(* Logix 5000 project; controller SX_V040001_C001 vendor 1 type 14 code 77 rev 16.22; software revision 16.04; part 6 of 35 *)
(* tags used below, declared in another part *)
   ALARM_BITS : INT[10];
   ALL_KINDS : INT[90];
   Basic : INT;
   G_DInput : DINT[3];
   G_DOutput : DINT[3];
   m_alarm_exist : BOOL;
   m_notstop : BOOL;
   METERING : INT[44];
   PARAMETER : INT[501];
   T_MET10_END : TIMER;
   T_MET11_END : TIMER;
   T_MET6_END : TIMER;
   T_MET7_END : TIMER;
   T_MET8_END : TIMER;
   T_MET9_END : TIMER;
   T_MET_VALVE_10 : TIMER;
   T_MET_VALVE_11 : TIMER;
   T_MET_VALVE_12 : TIMER;
   T_MET_VALVE_6 : TIMER;
   T_MET_VALVE_7 : TIMER;
   T_MET_VALVE_8 : TIMER;
   T_MET_VALVE_9 : TIMER;
   Z41 : COUNTER;
   Z42 : COUNTER;
   Z43 : COUNTER;
   Z44 : COUNTER;
   Z45 : COUNTER;
   Z46 : COUNTER;
   Z47 : COUNTER;
   Z48 : COUNTER;
   Z49 : COUNTER;
   Z50 : COUNTER;
(* MainProgram, continued *)

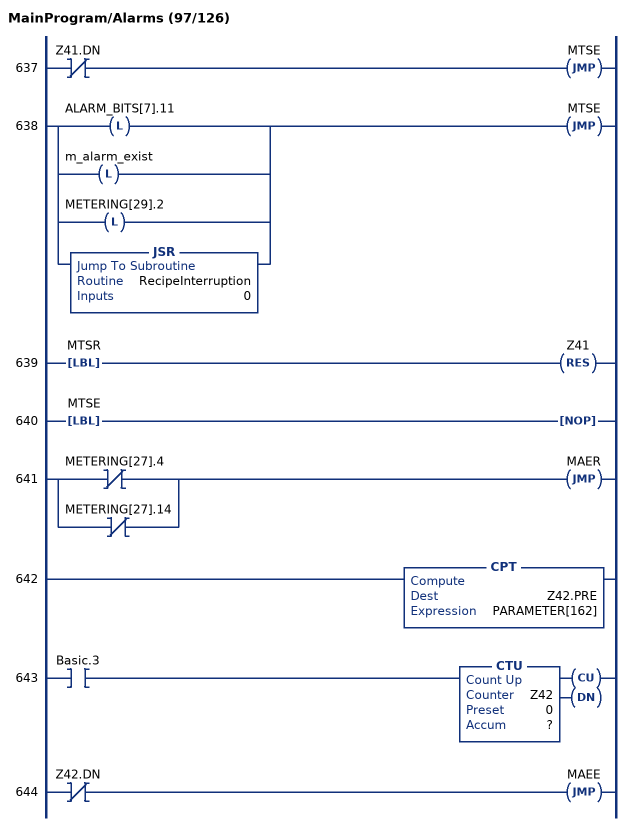
   [picture p118: MainProgram/Alarms rungs 637-644]
   637: XIO(Z41.DN)JMP(MTSE);
   638: [OTL(ALARM_BITS[7].11) ,OTL(m_alarm_exist) ,OTL(METERING[29].2) ,JSR(RecipeInterruption,0) ]JMP(MTSE);
   639: LBL(MTSR)RES(Z41);
   640: LBL(MTSE)NOP();
   641: [XIO(METERING[27].4) ,XIO(METERING[27].14) ]JMP(MAER);
   642: CPT(Z42.PRE,PARAMETER[162]);
   643: XIC(Basic.3)CTU(Z42,?,?);
   644: XIO(Z42.DN)JMP(MAEE);
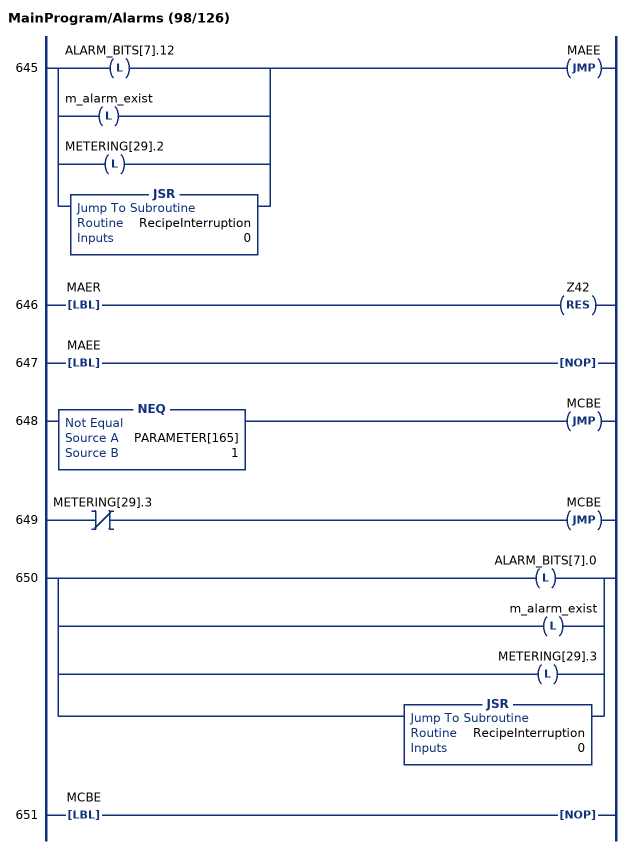
   645: [OTL(ALARM_BITS[7].12) ,OTL(m_alarm_exist) ,OTL(METERING[29].2) ,JSR(RecipeInterruption,0) ]JMP(MAEE);
   646: LBL(MAER)RES(Z42);
   647: LBL(MAEE)NOP();
   648: NEQ(PARAMETER[165],1)JMP(MCBE);
   649: XIO(METERING[29].3)JMP(MCBE);
   650: [OTL(ALARM_BITS[7].0) ,OTL(m_alarm_exist) ,OTL(METERING[29].3) ,JSR(RecipeInterruption,0) ];
   651: LBL(MCBE)NOP();
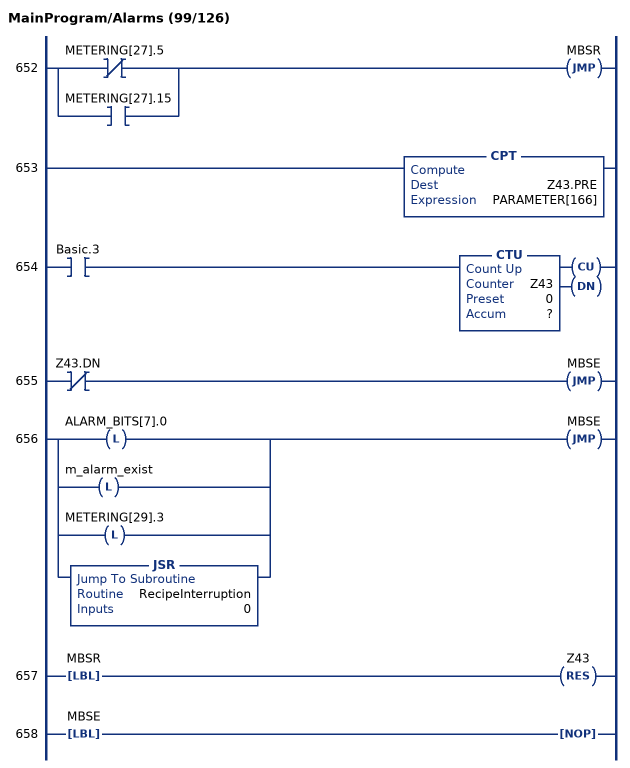
   652: [XIO(METERING[27].5) ,XIC(METERING[27].15) ]JMP(MBSR);
   653: CPT(Z43.PRE,PARAMETER[166]);
   654: XIC(Basic.3)CTU(Z43,?,?);
   655: XIO(Z43.DN)JMP(MBSE);
   656: [OTL(ALARM_BITS[7].0) ,OTL(m_alarm_exist) ,OTL(METERING[29].3) ,JSR(RecipeInterruption,0) ]JMP(MBSE);
   657: LBL(MBSR)RES(Z43);
   658: LBL(MBSE)NOP();
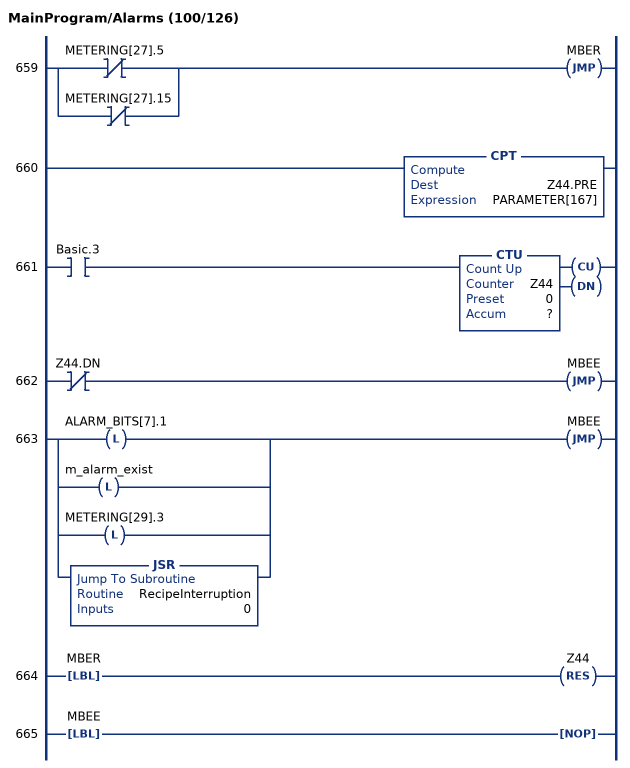
   659: [XIO(METERING[27].5) ,XIO(METERING[27].15) ]JMP(MBER);
   660: CPT(Z44.PRE,PARAMETER[167]);
   661: XIC(Basic.3)CTU(Z44,?,?);
   662: XIO(Z44.DN)JMP(MBEE);
   663: [OTL(ALARM_BITS[7].1) ,OTL(m_alarm_exist) ,OTL(METERING[29].3) ,JSR(RecipeInterruption,0) ]JMP(MBEE);
   664: LBL(MBER)RES(Z44);
   665: LBL(MBEE)NOP();
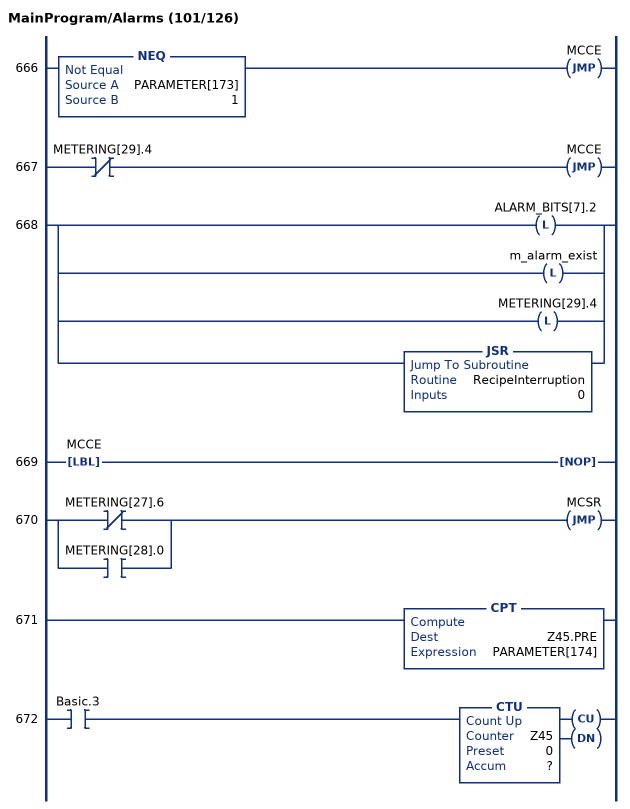
   666: NEQ(PARAMETER[173],1)JMP(MCCE);
   667: XIO(METERING[29].4)JMP(MCCE);
   668: [OTL(ALARM_BITS[7].2) ,OTL(m_alarm_exist) ,OTL(METERING[29].4) ,JSR(RecipeInterruption,0) ];
   669: LBL(MCCE)NOP();
   670: [XIO(METERING[27].6) ,XIC(METERING[28].0) ]JMP(MCSR);
   671: CPT(Z45.PRE,PARAMETER[174]);
   672: XIC(Basic.3)CTU(Z45,?,?);
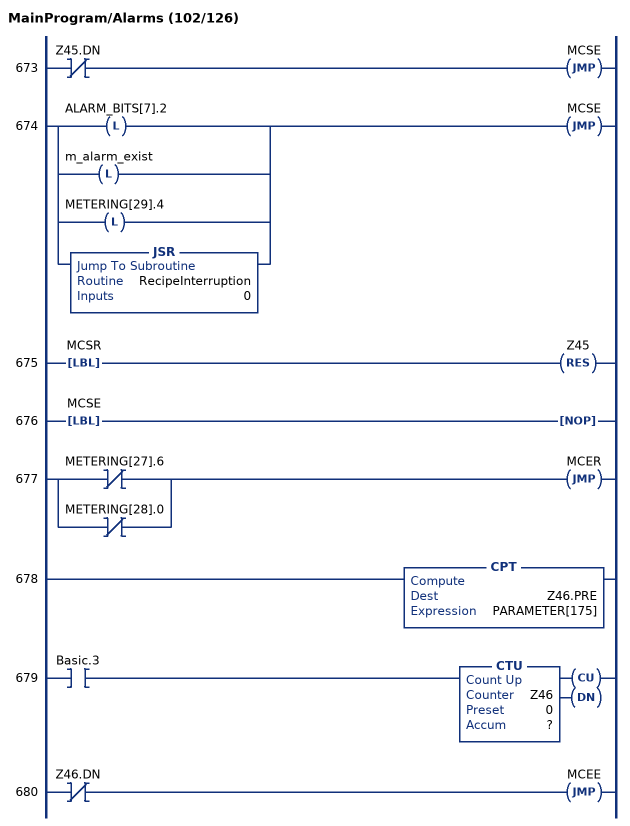
   673: XIO(Z45.DN)JMP(MCSE);
   674: [OTL(ALARM_BITS[7].2) ,OTL(m_alarm_exist) ,OTL(METERING[29].4) ,JSR(RecipeInterruption,0) ]JMP(MCSE);
   675: LBL(MCSR)RES(Z45);
   676: LBL(MCSE)NOP();
   677: [XIO(METERING[27].6) ,XIO(METERING[28].0) ]JMP(MCER);
   678: CPT(Z46.PRE,PARAMETER[175]);
   679: XIC(Basic.3)CTU(Z46,?,?);
   680: XIO(Z46.DN)JMP(MCEE);
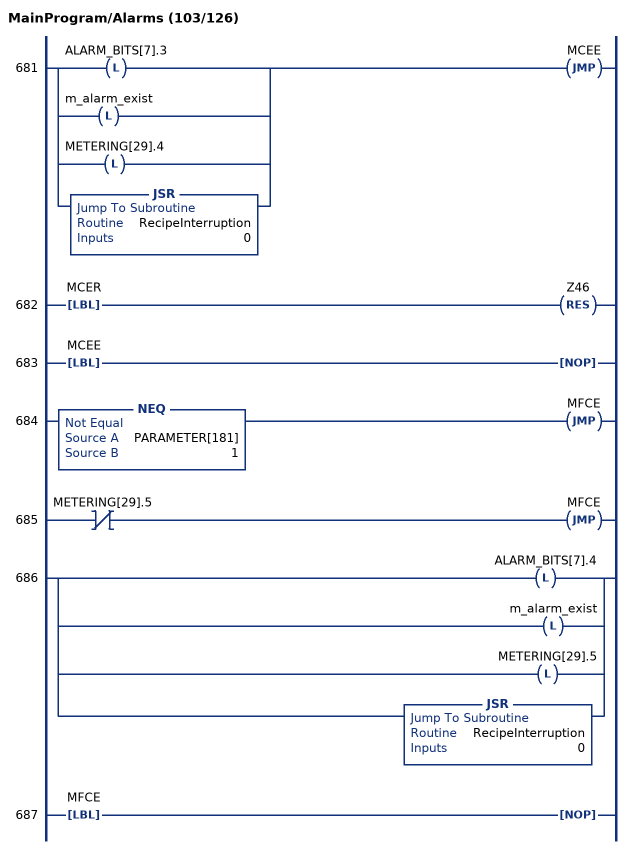
   681: [OTL(ALARM_BITS[7].3) ,OTL(m_alarm_exist) ,OTL(METERING[29].4) ,JSR(RecipeInterruption,0) ]JMP(MCEE);
   682: LBL(MCER)RES(Z46);
   683: LBL(MCEE)NOP();
   684: NEQ(PARAMETER[181],1)JMP(MFCE);
   685: XIO(METERING[29].5)JMP(MFCE);
   686: [OTL(ALARM_BITS[7].4) ,OTL(m_alarm_exist) ,OTL(METERING[29].5) ,JSR(RecipeInterruption,0) ];
   687: LBL(MFCE)NOP();
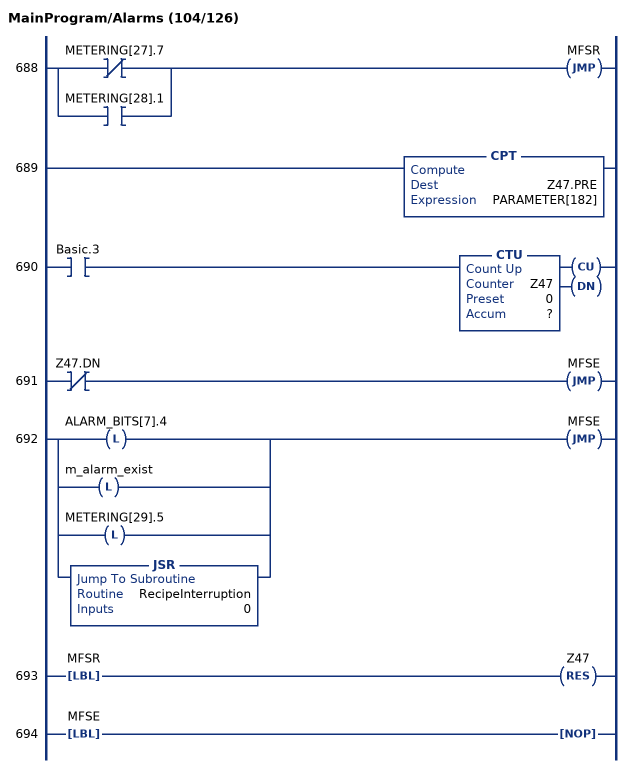
   688: [XIO(METERING[27].7) ,XIC(METERING[28].1) ]JMP(MFSR);
   689: CPT(Z47.PRE,PARAMETER[182]);
   690: XIC(Basic.3)CTU(Z47,?,?);
   691: XIO(Z47.DN)JMP(MFSE);
   692: [OTL(ALARM_BITS[7].4) ,OTL(m_alarm_exist) ,OTL(METERING[29].5) ,JSR(RecipeInterruption,0) ]JMP(MFSE);
   693: LBL(MFSR)RES(Z47);
   694: LBL(MFSE)NOP();
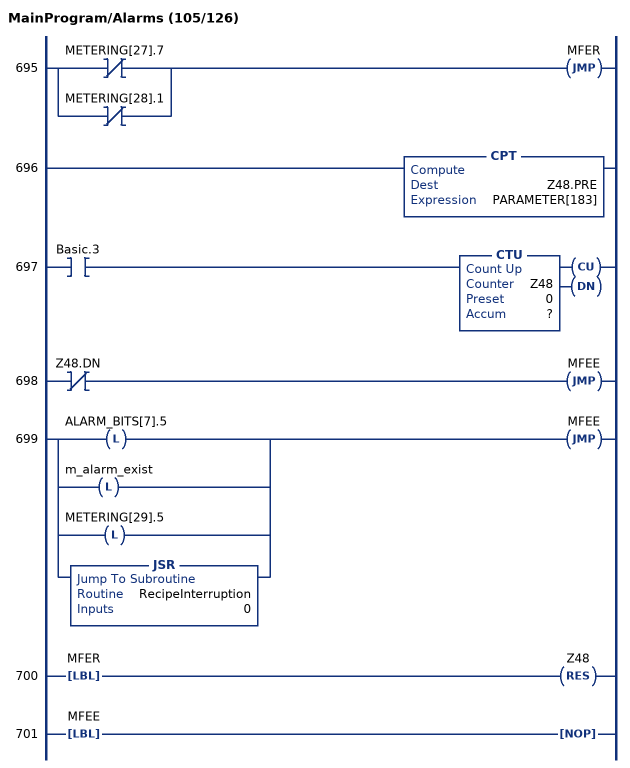
   695: [XIO(METERING[27].7) ,XIO(METERING[28].1) ]JMP(MFER);
   696: CPT(Z48.PRE,PARAMETER[183]);
   697: XIC(Basic.3)CTU(Z48,?,?);
   698: XIO(Z48.DN)JMP(MFEE);
   699: [OTL(ALARM_BITS[7].5) ,OTL(m_alarm_exist) ,OTL(METERING[29].5) ,JSR(RecipeInterruption,0) ]JMP(MFEE);
   700: LBL(MFER)RES(Z48);
   701: LBL(MFEE)NOP();
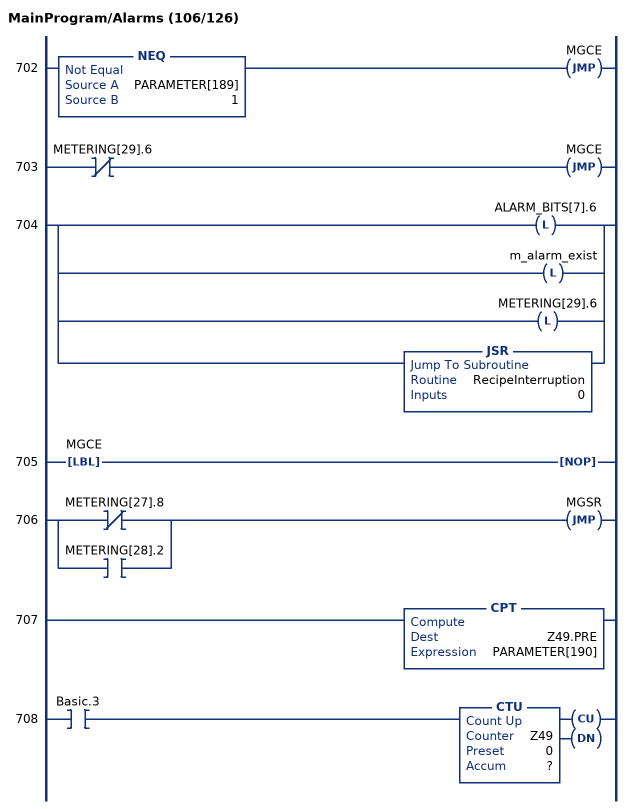
   702: NEQ(PARAMETER[189],1)JMP(MGCE);
   703: XIO(METERING[29].6)JMP(MGCE);
   704: [OTL(ALARM_BITS[7].6) ,OTL(m_alarm_exist) ,OTL(METERING[29].6) ,JSR(RecipeInterruption,0) ];
   705: LBL(MGCE)NOP();
   706: [XIO(METERING[27].8) ,XIC(METERING[28].2) ]JMP(MGSR);
   707: CPT(Z49.PRE,PARAMETER[190]);
   708: XIC(Basic.3)CTU(Z49,?,?);
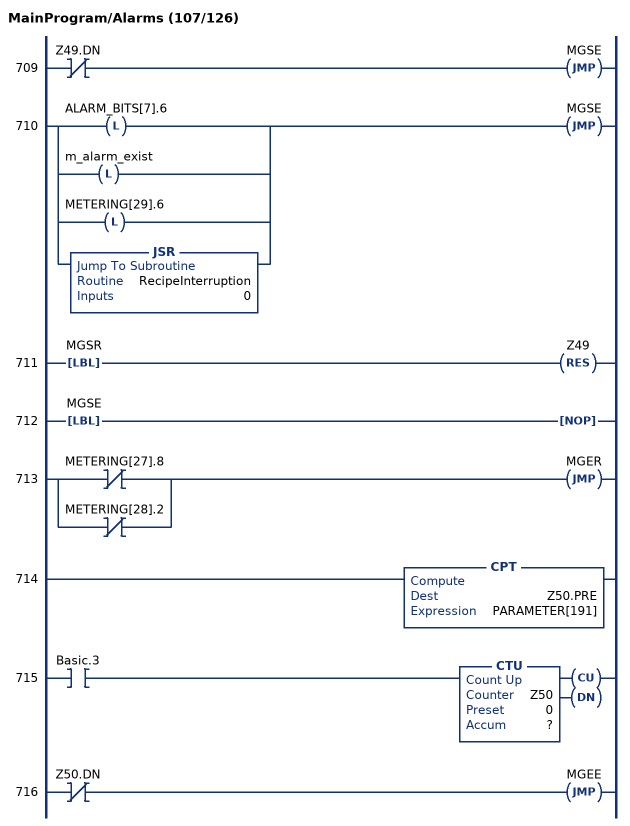
   709: XIO(Z49.DN)JMP(MGSE);
   710: [OTL(ALARM_BITS[7].6) ,OTL(m_alarm_exist) ,OTL(METERING[29].6) ,JSR(RecipeInterruption,0) ]JMP(MGSE);
   711: LBL(MGSR)RES(Z49);
   712: LBL(MGSE)NOP();
   713: [XIO(METERING[27].8) ,XIO(METERING[28].2) ]JMP(MGER);
   714: CPT(Z50.PRE,PARAMETER[191]);
   715: XIC(Basic.3)CTU(Z50,?,?);
   716: XIO(Z50.DN)JMP(MGEE);
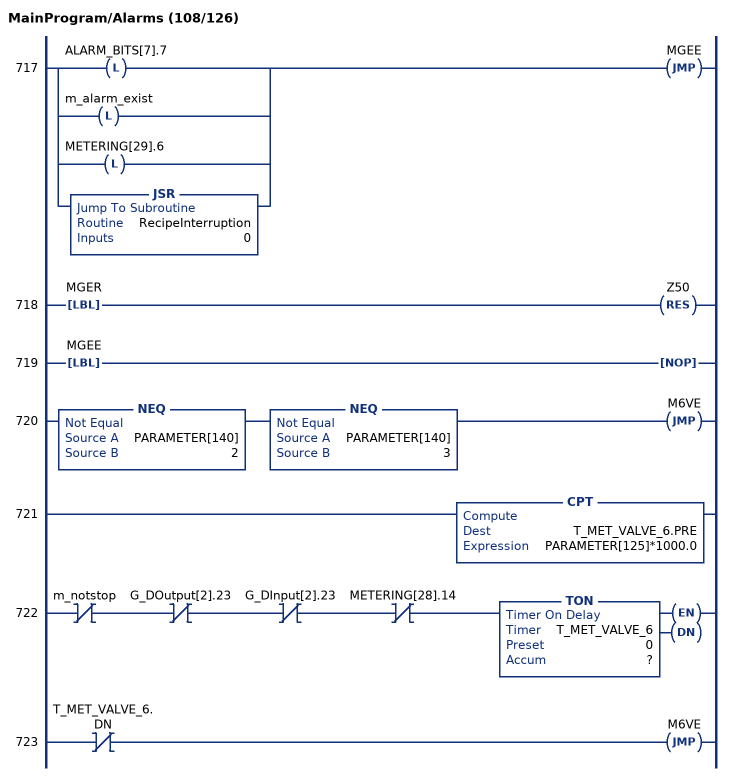
   717: [OTL(ALARM_BITS[7].7) ,OTL(m_alarm_exist) ,OTL(METERING[29].6) ,JSR(RecipeInterruption,0) ]JMP(MGEE);
   718: LBL(MGER)RES(Z50);
   719: LBL(MGEE)NOP();
   720: NEQ(PARAMETER[140],2)NEQ(PARAMETER[140],3)JMP(M6VE);
   721: CPT(T_MET_VALVE_6.PRE,PARAMETER[125]*1000.0);
   722: XIO(m_notstop)XIO(G_DOutput[2].23)XIO(G_DInput[2].23)XIO(METERING[28].14)TON(T_MET_VALVE_6,?,?);
   723: XIO(T_MET_VALVE_6.DN)JMP(M6VE);
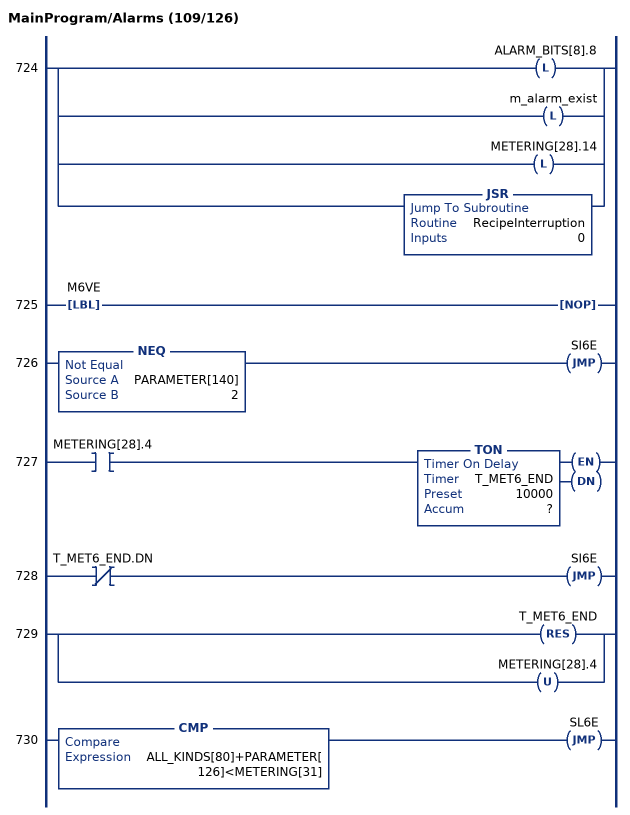
   724: [OTL(ALARM_BITS[8].8) ,OTL(m_alarm_exist) ,OTL(METERING[28].14) ,JSR(RecipeInterruption,0) ];
   725: LBL(M6VE)NOP();
   726: NEQ(PARAMETER[140],2)JMP(SI6E);
   727: XIC(METERING[28].4)TON(T_MET6_END,?,?);
   728: XIO(T_MET6_END.DN)JMP(SI6E);
   729: [RES(T_MET6_END) ,OTU(METERING[28].4) ];
   730: CMP(ALL_KINDS[80]+PARAMETER[126]<METERING[31])JMP(SL6E);
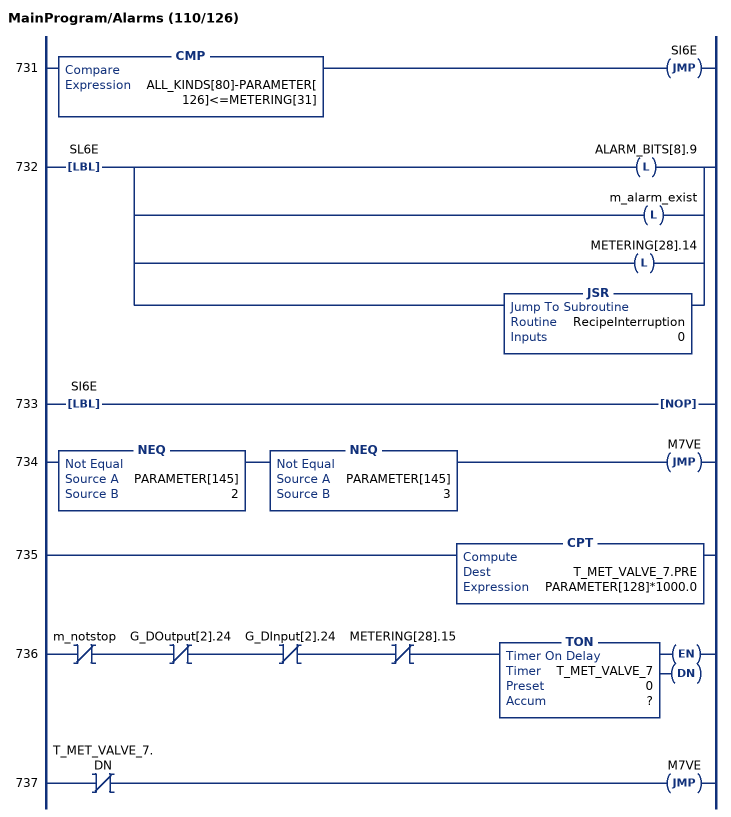
   731: CMP(ALL_KINDS[80]-PARAMETER[126]<=METERING[31])JMP(SI6E);
   732: LBL(SL6E)[OTL(ALARM_BITS[8].9) ,OTL(m_alarm_exist) ,OTL(METERING[28].14) ,JSR(RecipeInterruption,0) ];
   733: LBL(SI6E)NOP();
   734: NEQ(PARAMETER[145],2)NEQ(PARAMETER[145],3)JMP(M7VE);
   735: CPT(T_MET_VALVE_7.PRE,PARAMETER[128]*1000.0);
   736: XIO(m_notstop)XIO(G_DOutput[2].24)XIO(G_DInput[2].24)XIO(METERING[28].15)TON(T_MET_VALVE_7,?,?);
   737: XIO(T_MET_VALVE_7.DN)JMP(M7VE);
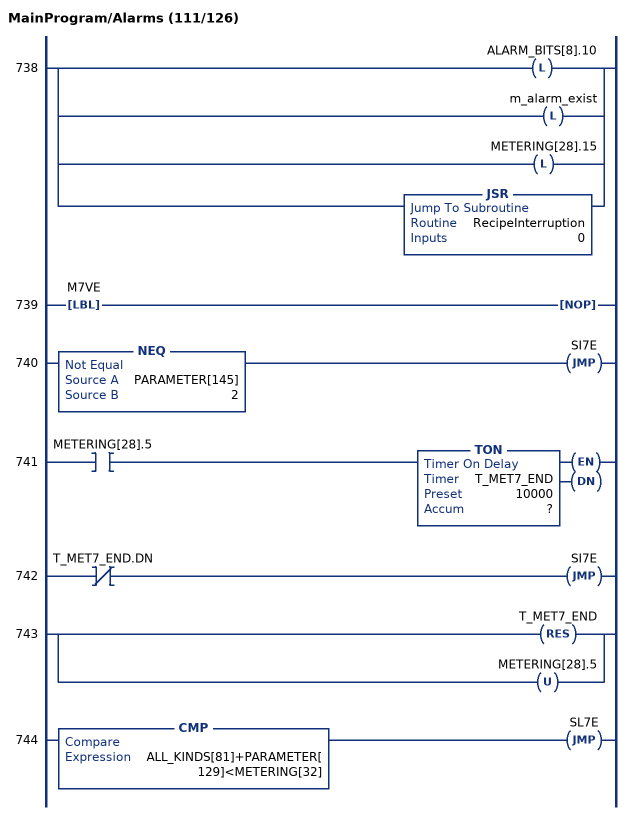
   738: [OTL(ALARM_BITS[8].10) ,OTL(m_alarm_exist) ,OTL(METERING[28].15) ,JSR(RecipeInterruption,0) ];
   739: LBL(M7VE)NOP();
   740: NEQ(PARAMETER[145],2)JMP(SI7E);
   741: XIC(METERING[28].5)TON(T_MET7_END,?,?);
   742: XIO(T_MET7_END.DN)JMP(SI7E);
   743: [RES(T_MET7_END) ,OTU(METERING[28].5) ];
   744: CMP(ALL_KINDS[81]+PARAMETER[129]<METERING[32])JMP(SL7E);
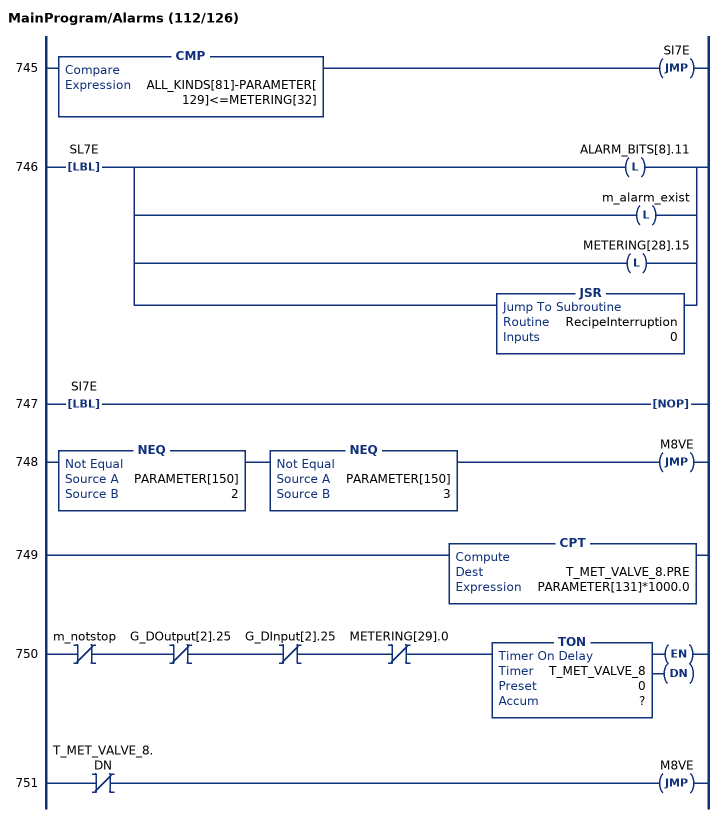
   745: CMP(ALL_KINDS[81]-PARAMETER[129]<=METERING[32])JMP(SI7E);
   746: LBL(SL7E)[OTL(ALARM_BITS[8].11) ,OTL(m_alarm_exist) ,OTL(METERING[28].15) ,JSR(RecipeInterruption,0) ];
   747: LBL(SI7E)NOP();
   748: NEQ(PARAMETER[150],2)NEQ(PARAMETER[150],3)JMP(M8VE);
   749: CPT(T_MET_VALVE_8.PRE,PARAMETER[131]*1000.0);
   750: XIO(m_notstop)XIO(G_DOutput[2].25)XIO(G_DInput[2].25)XIO(METERING[29].0)TON(T_MET_VALVE_8,?,?);
   751: XIO(T_MET_VALVE_8.DN)JMP(M8VE);
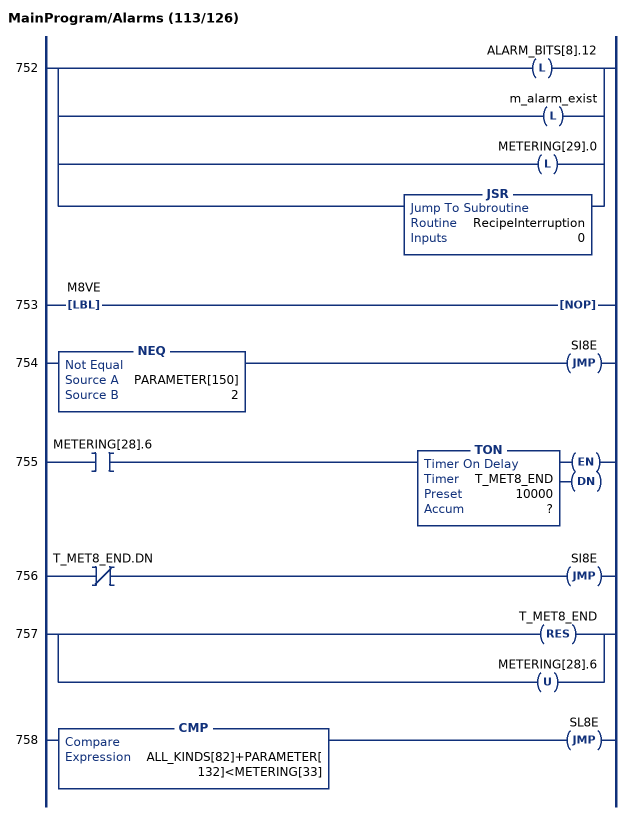
   752: [OTL(ALARM_BITS[8].12) ,OTL(m_alarm_exist) ,OTL(METERING[29].0) ,JSR(RecipeInterruption,0) ];
   753: LBL(M8VE)NOP();
   754: NEQ(PARAMETER[150],2)JMP(SI8E);
   755: XIC(METERING[28].6)TON(T_MET8_END,?,?);
   756: XIO(T_MET8_END.DN)JMP(SI8E);
   757: [RES(T_MET8_END) ,OTU(METERING[28].6) ];
   758: CMP(ALL_KINDS[82]+PARAMETER[132]<METERING[33])JMP(SL8E);
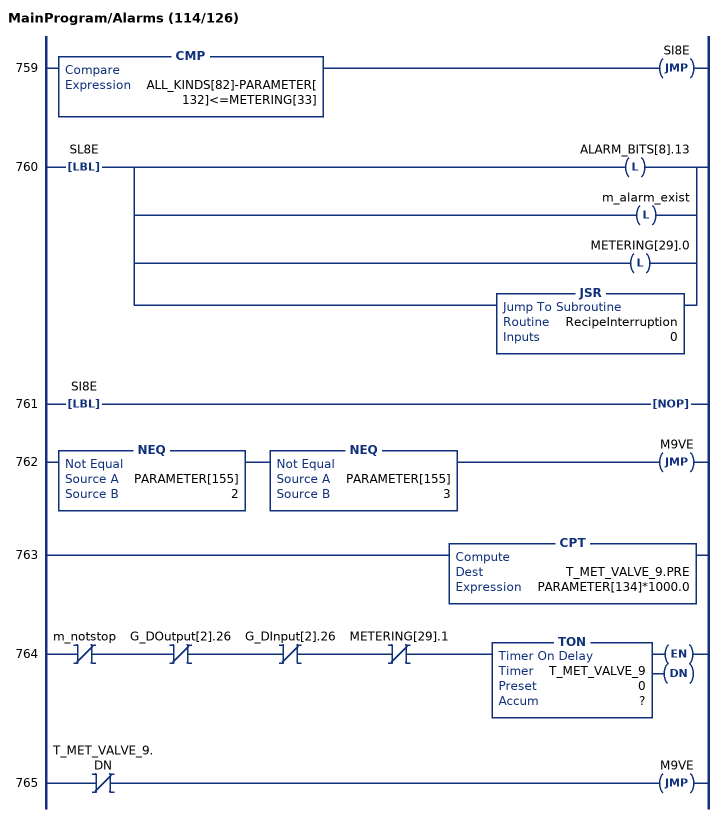
   759: CMP(ALL_KINDS[82]-PARAMETER[132]<=METERING[33])JMP(SI8E);
   760: LBL(SL8E)[OTL(ALARM_BITS[8].13) ,OTL(m_alarm_exist) ,OTL(METERING[29].0) ,JSR(RecipeInterruption,0) ];
   761: LBL(SI8E)NOP();
   762: NEQ(PARAMETER[155],2)NEQ(PARAMETER[155],3)JMP(M9VE);
   763: CPT(T_MET_VALVE_9.PRE,PARAMETER[134]*1000.0);
   764: XIO(m_notstop)XIO(G_DOutput[2].26)XIO(G_DInput[2].26)XIO(METERING[29].1)TON(T_MET_VALVE_9,?,?);
   765: XIO(T_MET_VALVE_9.DN)JMP(M9VE);
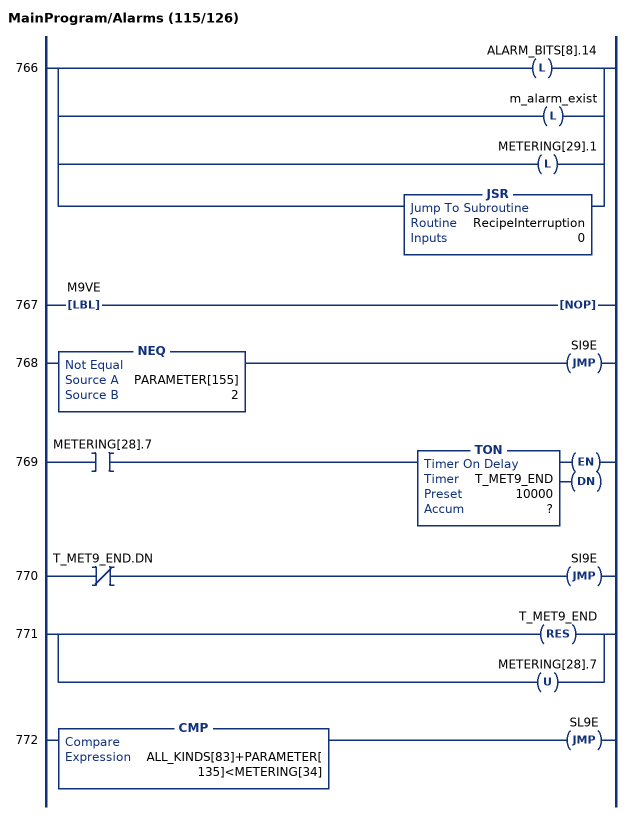
   766: [OTL(ALARM_BITS[8].14) ,OTL(m_alarm_exist) ,OTL(METERING[29].1) ,JSR(RecipeInterruption,0) ];
   767: LBL(M9VE)NOP();
   768: NEQ(PARAMETER[155],2)JMP(SI9E);
   769: XIC(METERING[28].7)TON(T_MET9_END,?,?);
   770: XIO(T_MET9_END.DN)JMP(SI9E);
   771: [RES(T_MET9_END) ,OTU(METERING[28].7) ];
   772: CMP(ALL_KINDS[83]+PARAMETER[135]<METERING[34])JMP(SL9E);
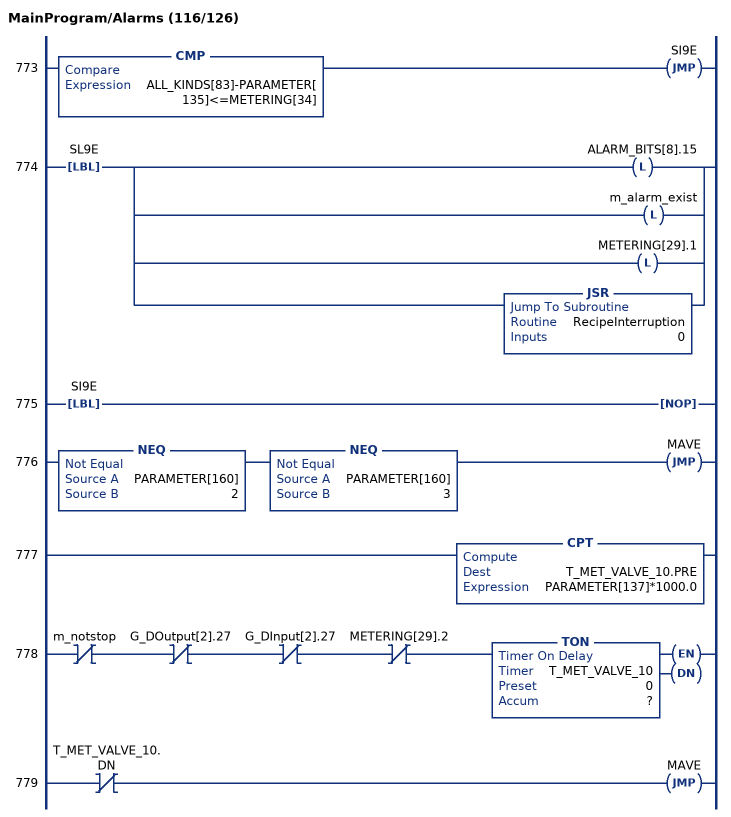
   773: CMP(ALL_KINDS[83]-PARAMETER[135]<=METERING[34])JMP(SI9E);
   774: LBL(SL9E)[OTL(ALARM_BITS[8].15) ,OTL(m_alarm_exist) ,OTL(METERING[29].1) ,JSR(RecipeInterruption,0) ];
   775: LBL(SI9E)NOP();
   776: NEQ(PARAMETER[160],2)NEQ(PARAMETER[160],3)JMP(MAVE);
   777: CPT(T_MET_VALVE_10.PRE,PARAMETER[137]*1000.0);
   778: XIO(m_notstop)XIO(G_DOutput[2].27)XIO(G_DInput[2].27)XIO(METERING[29].2)TON(T_MET_VALVE_10,?,?);
   779: XIO(T_MET_VALVE_10.DN)JMP(MAVE);
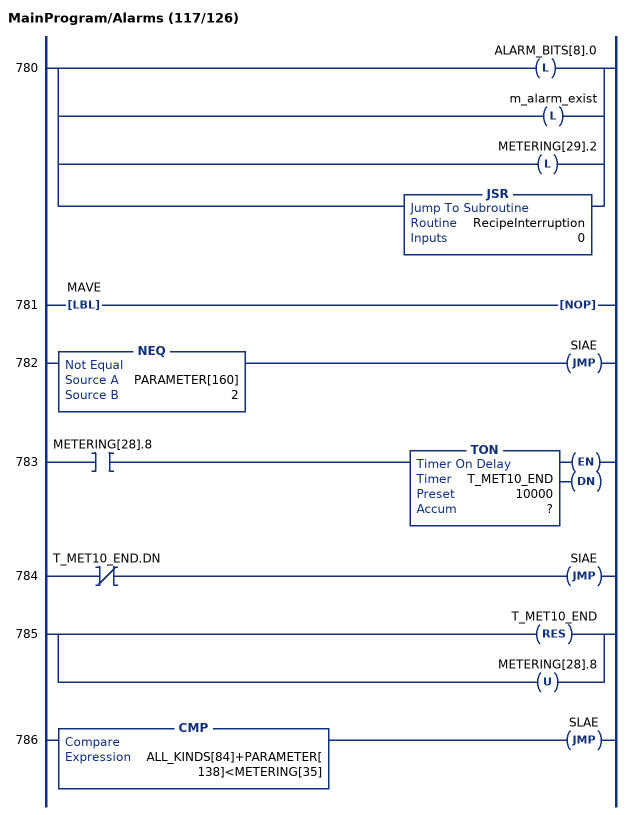
   780: [OTL(ALARM_BITS[8].0) ,OTL(m_alarm_exist) ,OTL(METERING[29].2) ,JSR(RecipeInterruption,0) ];
   781: LBL(MAVE)NOP();
   782: NEQ(PARAMETER[160],2)JMP(SIAE);
   783: XIC(METERING[28].8)TON(T_MET10_END,?,?);
   784: XIO(T_MET10_END.DN)JMP(SIAE);
   785: [RES(T_MET10_END) ,OTU(METERING[28].8) ];
   786: CMP(ALL_KINDS[84]+PARAMETER[138]<METERING[35])JMP(SLAE);
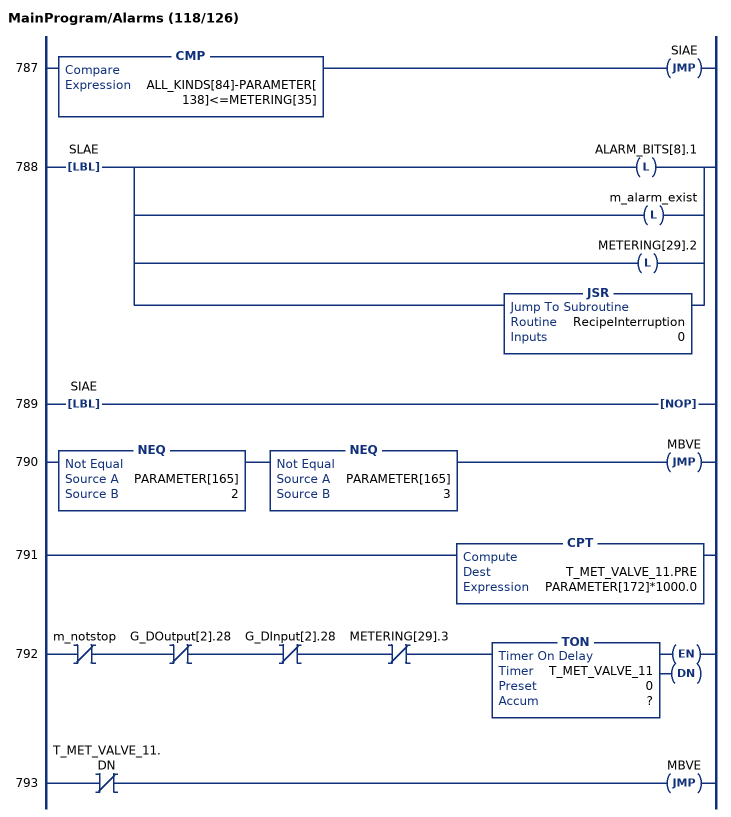
   787: CMP(ALL_KINDS[84]-PARAMETER[138]<=METERING[35])JMP(SIAE);
   788: LBL(SLAE)[OTL(ALARM_BITS[8].1) ,OTL(m_alarm_exist) ,OTL(METERING[29].2) ,JSR(RecipeInterruption,0) ];
   789: LBL(SIAE)NOP();
   790: NEQ(PARAMETER[165],2)NEQ(PARAMETER[165],3)JMP(MBVE);
   791: CPT(T_MET_VALVE_11.PRE,PARAMETER[172]*1000.0);
   792: XIO(m_notstop)XIO(G_DOutput[2].28)XIO(G_DInput[2].28)XIO(METERING[29].3)TON(T_MET_VALVE_11,?,?);
   793: XIO(T_MET_VALVE_11.DN)JMP(MBVE);
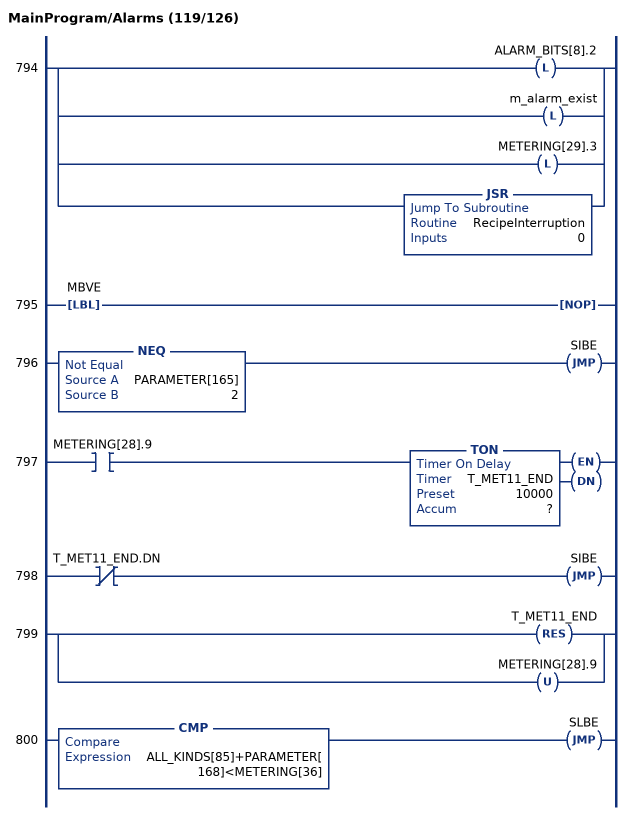
   794: [OTL(ALARM_BITS[8].2) ,OTL(m_alarm_exist) ,OTL(METERING[29].3) ,JSR(RecipeInterruption,0) ];
   795: LBL(MBVE)NOP();
   796: NEQ(PARAMETER[165],2)JMP(SIBE);
   797: XIC(METERING[28].9)TON(T_MET11_END,?,?);
   798: XIO(T_MET11_END.DN)JMP(SIBE);
   799: [RES(T_MET11_END) ,OTU(METERING[28].9) ];
   800: CMP(ALL_KINDS[85]+PARAMETER[168]<METERING[36])JMP(SLBE);
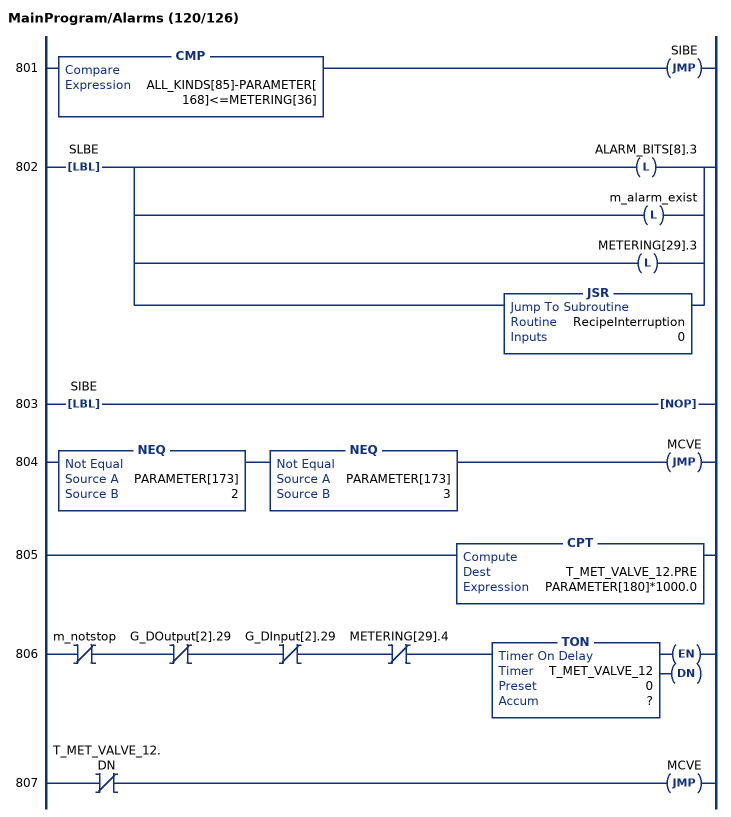
   801: CMP(ALL_KINDS[85]-PARAMETER[168]<=METERING[36])JMP(SIBE);
   802: LBL(SLBE)[OTL(ALARM_BITS[8].3) ,OTL(m_alarm_exist) ,OTL(METERING[29].3) ,JSR(RecipeInterruption,0) ];
   803: LBL(SIBE)NOP();
   804: NEQ(PARAMETER[173],2)NEQ(PARAMETER[173],3)JMP(MCVE);
   805: CPT(T_MET_VALVE_12.PRE,PARAMETER[180]*1000.0);
   806: XIO(m_notstop)XIO(G_DOutput[2].29)XIO(G_DInput[2].29)XIO(METERING[29].4)TON(T_MET_VALVE_12,?,?);
   807: XIO(T_MET_VALVE_12.DN)JMP(MCVE);
